(* PLC project CoDeSys External Library Template, WAGO e!COCKPIT e!COCKPIT, author 3S - Smart Software Solutions GmbH *)
(* stored: creationDateTime 2019-10-29T12:37:19.9643048, version 3.5.5.30, modificationDateTime 2019-10-29T12:36:39.3744516, organization 3S - Smart Software Solutions GmbH *)
(* Library project template with all possible element types, docu and a sample project structure *)

FUNCTION fnRozbicieNaBityRejestru16Bit : BOOL
  VAR_INPUT
    wRejestr16Bit : WORD;
  END_VAR
  VAR_OUTPUT
    xBit0 : BOOL;
    xBit1 : BOOL;
    xBit2 : BOOL;
    xBit3 : BOOL;
    xBit4 : BOOL;
    xBit5 : BOOL;
    xBit6 : BOOL;
    xBit7 : BOOL;
    xBit8 : BOOL;
    xBit9 : BOOL;
    xBit10 : BOOL;
    xBit11 : BOOL;
    xBit12 : BOOL;
    xBit13 : BOOL;
    xBit14 : BOOL;
    xBit15 : BOOL;
  END_VAR
  VAR
    wTempRejestr16 : WORD;
  END_VAR

            (*			
Autor:					Paweł Kąkol, 
Prawa majątkowe: 		Solwena Sp. z o.o., 
Aktualizacje:			2017-11-17-10:00-PK

Opis:					Funkcja do rozbijania rejestru 16-bitowego typu WORD na pojedyncze zmienne BOOL,
						Nalezy pamietac, ze numeracja bitow jest zgodna z odpowiadajacymi wykladnikami potegi liczby 2
*)
wTempRejestr16 := wRejestr16Bit;
//sprawdzanie stanu bitow
IF wTempRejestr16 >= 32768 THEN
	xBit15 := TRUE;
	wTempRejestr16 := wTempRejestr16 MOD 32768;
ELSE
	xBit15 := FALSE;	
END_IF
IF wTempRejestr16 >= 16384 THEN
	xBit14 := TRUE;
	wTempRejestr16 := wTempRejestr16 MOD 16384;
ELSE
	xBit14 := FALSE;
END_IF
IF wTempRejestr16 >= 8192 THEN
	xBit13 := TRUE;
	wTempRejestr16 := wTempRejestr16 MOD 8192;
ELSE
	xBit13 := FALSE;
END_IF
IF wTempRejestr16 >= 4096 THEN
	xBit12 := TRUE;
	wTempRejestr16 := wTempRejestr16 MOD 4096;
ELSE
	xBit12 := FALSE;
END_IF
IF wTempRejestr16 >= 2048 THEN
	xBit11 := TRUE;
	wTempRejestr16 := wTempRejestr16 MOD 2048;
ELSE
	xBit11 := FALSE;
END_IF
IF wTempRejestr16 >= 1024 THEN
	xBit10 := TRUE;
	wTempRejestr16 := wTempRejestr16 MOD 1024;
ELSE
	xBit10 := FALSE;
END_IF
IF wTempRejestr16 >= 512 THEN
	xBit9 := TRUE;
	wTempRejestr16 := wTempRejestr16 MOD 512;
ELSE
	xBit9 := FALSE;
END_IF
IF wTempRejestr16 >= 256 THEN
	xBit8 := TRUE;
	wTempRejestr16 := wTempRejestr16 MOD 256;
ELSE
	xBit8 := FALSE;
END_IF
IF wTempRejestr16 >= 128 THEN
	xBit7 := TRUE;
	wTempRejestr16 := wTempRejestr16 MOD 128;
ELSE
	xBit7 := FALSE;
END_IF
IF wTempRejestr16 >= 64 THEN
	xBit6 := TRUE;
	wTempRejestr16 := wTempRejestr16 MOD 64;
ELSE
	xBit6 := FALSE;
END_IF
IF wTempRejestr16 >= 32 THEN
	xBit5 := TRUE;
	wTempRejestr16 := wTempRejestr16 MOD 32;
ELSE
	xBit5 := FALSE;
END_IF
IF wTempRejestr16 >= 16 THEN
	xBit4 := TRUE;
	wTempRejestr16 := wTempRejestr16 MOD 16;
ELSE
	xBit4 := FALSE;
END_IF
IF wTempRejestr16 >= 8 THEN
	xBit3 := TRUE;
	wTempRejestr16 := wTempRejestr16 MOD 8;
ELSE
	xBit3 := FALSE;
END_IF
IF wTempRejestr16 >= 4 THEN
	xBit2 := TRUE;
	wTempRejestr16 := wTempRejestr16 MOD 4;
ELSE
	xBit2 := FALSE;
END_IF
IF wTempRejestr16 >= 2 THEN
	xBit1 := TRUE;
	wTempRejestr16 := wTempRejestr16 MOD 2;
ELSE
	xBit1 := FALSE;
END_IF
IF wTempRejestr16 >= 1 THEN
	xBit0 := TRUE;
ELSE
	xBit0 := FALSE;
END_IF
          
END_FUNCTION
